(* CODESYS project SingleAxis.export

Project tree, tasks and I/O mapping:
  program SingleAxis [ST]
*)

// SingleAxis
PROGRAM SingleAxis
VAR
	Enable : BOOL;
	StartMov : BOOL;
	MovAxis : INT := 0;
	FirstPos : REAL := -180;
	SecondPos : REAL := 180;
	CurrentPos : REAL;
	Vel : REAL := 180;
	Acc : REAL := 180;
	Jerk : REAL := 180;
	stopTime : TIME := T#1S;
	MovErr : BOOL;
	
	PowBlk : ArcaLibrary.MC_Power;
	PowDone, PowErr : BOOL;
	
	MovState : INT;
	FirMov : ArcaLibrary.MC_MoveAbsolute;
	SecMov : ArcaLibrary.MC_MoveAbsolute;
	StopMov : ArcaLibrary.MC_Stop;
	dis_trig : r_trig;
	
	ReadPos : ArcaLibrary.MCAT_ReadAxisMeasures;
	StopTimer : ton;
END_VAR


PowBlk(Axis := MovAxis, Enable:=Enable, EnablePositive:=TRUE, EnableNegative:=TRUE, Status=>PowDone, Error=>PowErr);
ReadPos(axis := MovAxis, enable := PowBlk.Status, pos=> currentPos);

dis_trig(clk := NOT startMov);
StopMov(axis := MovAxis, execute := dis_trig.Q, Deceleration := acc*10, jerk := jerk*10);

IF MovState > 20 AND NOT startMov THEN
	MovState := 20;
END_IF
CASE MovState OF
	0:
		IF PowDone THEN
			MovState := 10;
		END_IF
	10:
		IF startMov THEN
			MovState := 20;
		END_IF
	20:
		FirMov(axis := MovAxis, Execute := FALSE);
		SecMov(axis := MovAxis, Execute := FALSE);
		IF startMov THEN
			StopTimer(in:= FALSE);
			MovState := 30;
		ELSE
			MovState := 0;
		END_IF
	30:
		FirMov(axis := MovAxis, Execute := TRUE, Position := FirstPos
			, Velocity := vel, Acceleration := acc, Deceleration := Acc, jerk := jerk
			, Direction := mcShortestWay, BufferMode := mcAborting 
			, Error => MovErr);
		IF FirMov.Done THEN
			IF stopTime > T#0S THEN
			StopTimer (in := TRUE, PT := stopTime);
				MovState := 35;
			ELSE
				MovState := 40;
			END_IF
		END_IF
	35:
		StopTimer (in := TRUE, PT := stopTime);
		IF StopTimer.Q THEN
			StopTimer(in:= FALSE);
			MovState := 40;
		END_IF
	40:
		SecMov(axis := MovAxis, Execute := TRUE, Position := SecondPos
			, Velocity := vel, Acceleration := acc, Deceleration := Acc, jerk := jerk
			, Direction := mcShortestWay, BufferMode := mcAborting 
			, Error => MovErr);
		IF SecMov.Done THEN
			StopTimer (in := TRUE, PT := stopTime);
			IF stopTime > T#0S THEN
				MovState := 45;
			ELSE
			MovState := 20;
			END_IF
		END_IF
	45:
		StopTimer (in := TRUE, PT := stopTime);
		IF StopTimer.Q THEN
			StopTimer(in:= FALSE);
			MovState := 20;
		END_IF
END_CASE

END_PROGRAM
